TYPE EL3152_DEV_STATUS :
    STRUCT
      
		Underrange : BOOL;
		Overrange : BOOL;
		Limit1 : BOOL;
		Limit2 : BOOL;
		Error : BOOL;
		TxPDOState : BOOL;
		TxPDOToggle : BOOL;
	
    END_STRUCT
END_TYPE

(* stored: Version 1.1.0.1, ProductVersion 3.1.4024.15
   DUT EL3152_DEV_STATUS: Id {b4407ae8-c4d4-4bab-bc9f-67e131f91519} *)
